Fanuc KAREL source: kt00153.KL

-- PROVISIONAL review KL for V1013-1; original PC SHA256 5b68402e9c74a46cb97ab7b1f873c76de1e8aedd5e62ac0c5507893227b317fd
-- Incomplete behavior may be omitted. Consult companion uncertainty JSON. Do not deploy.
PROGRAM KT00153
%NOLOCKGROUP
VAR
  I2 : INTEGER
  OUT : INTEGER
-- UNRESOLVED_DECL H1 type=002017
BEGIN
  -- UNRESOLVED_PC offsets 5-19; opcodes 2E,22,9D,33,B4
  -- UNRESOLVED_PC offsets 24-35; opcodes 2E,23
  -- UNRESOLVED_PC offsets 40-62; opcodes 22,9D,33,B3,21,55,23
  -- UNRESOLVED_PC offsets 67-71; opcodes 7F
END KT00153
